FUNCTION FAILED_AND_NOT_PENDING : BOOL
VAR_INPUT
	hr 	: DINT;
END_VAR
VAR
END_VAR

FAILED_AND_NOT_PENDING := hr <> S_OK AND hr <> S_PENDING;

END_FUNCTION

(* stored: Version 1.1.0.1, ProductVersion 3.1.4026.18
   POU FAILED_AND_NOT_PENDING: Id {c2668650-5b12-4634-9188-91a1822e5236}, SpecialFunc None *)
